PROGRAM CreateBasin
VAR
	state	:INT	:= 0;
END_VAR

CASE state OF
	0: //x min
	IF GVL_MOTION.EXT_CTR.BASINCTR THEN
		GVL_MOTION.EXT_CTR.BASINCTR			:= FALSE;
		GVL_MOTION.STATUS.BasinSet			:= FALSE;
		GVL_MOTION.STATUS.Basin_Set_Err		:= FALSE;
		IF GVL_MOTION.Basin.xMin >= GVL_MOTION.CARRIAGE_OFFSETS[0] THEN
			state							:= 1;
		ELSE
			GVL_MOTION.STATUS.Basin_Set_Err	:= TRUE;	
		END_IF
		
		
	ELSIF GVL_MOTION.EXT_CTR.DEFAULTBASIN THEN
		GVL_MOTION.EXT_CTR.DEFAULTBASIN		:= FALSE;
		GVL_MOTION.STATUS.Basin_Set_Err		:= FALSE;
		
		GVL_MOTION.Basin.xMin				:= GVL_MOTION.CARRIAGE_OFFSETS[0];
		GVL_MOTION.Basin.xMax				:= GVL_MOTION.STATUS.HardStopLocations[0];
		GVL_MOTION.Basin.yMin				:= GVL_MOTION.CARRIAGE_OFFSETS[1];
		GVL_MOTION.Basin.yMax				:= GVL_MOTION.STATUS.HardStopLocations[1];
		GVL_MOTION.Basin.Name				:= 'Full_Area';
		GVL_MOTION.STATUS.BasinSet			:= TRUE;
	END_IF
	
	1: //x max
		IF GVL_MOTION.Basin.xMax <= GVL_MOTION.STATUS.HardStopLocations[0] THEN
			state							:= 2;
		ELSE
			GVL_MOTION.STATUS.Basin_Set_Err	:= TRUE;
			state							:= 0;
		END_IF	
		
	
	2: //y min
	IF GVL_MOTION.Basin.yMin >= GVL_MOTION.CARRIAGE_OFFSETS[1] THEN
		state								:= 3;
	ELSE	
		GVL_MOTION.STATUS.Basin_Set_Err		:= TRUE;
		state								:= 0;
	END_IF
	
	3: //y max
	IF GVL_MOTION.Basin.yMax <= GVL_MOTION.STATUS.HardStopLocations[1] THEN
		state								:= 4;
	ELSE
		GVL_MOTION.STATUS.Basin_Set_Err		:= TRUE;
		state								:= 0;
	END_IF	

	
	4: //name
	IF GVL_MOTION.EXT_CTR.BASINNAME <> '' THEN
		GVL_MOTION.Basin.Name			:= GVL_MOTION.EXT_CTR.BASINNAME;
	ELSE
		GVL_MOTION.STATUS.Basin_Set_Err	:= TRUE;
	END_IF	
	state								:= 0;
END_CASE

END_PROGRAM

(* stored: Version 1.1.0.1, ProductVersion 3.1.4026.12
   POU CreateBasin: Id {d0232615-ad9b-44bb-bd96-662b703124b8}, SpecialFunc None *)
